TYPE String2Byte :
UNION
	sValue			:STRING; 
	arrByte 		:ARRAY[0..255] OF BYTE;
END_UNION
END_TYPE

(* stored: Version 1.1.0.1
   DUT String2Byte: Id {61023c66-9a3e-44c4-b77a-adb7c1c9bf66} *)
